// TIA Portal V20 export
// export: Created 2025-12-01T14:56:54.8600917Z, ExportSetting None, DisplayName Totally Integrated Automation Portal, DisplayVersion V20 Update 3, DisplayName TIA Portal Openness, DisplayVersion V20 Update 3, DisplayName TIA Portal Version Control Interface, DisplayVersion V20 Update 3, DisplayName STEP 7 Professional, DisplayVersion V20 Update 3, DisplayName STEP 7 Safety, DisplayVersion V20 Update 2, DisplayName WinCC Basic/Comfort/Advanced, DisplayVersion V20 Update 3, DisplayName WinCC Professional, DisplayVersion V20 Update 3, DisplayName WinCC Unified, DisplayVersion V20 Update 3
FUNCTION_BLOCK "FB343_ApiladorBandejas_RIANTICS"   // FB343, LAD
{ S7_Optimized_Access := 'FALSE' }
// stored: AutoNumber false, SetENOAutomatically false
   VAR_INPUT
      Maquina : UInt;   // Numero de Maquina (Mesa)
      Error_Tx : Bool;   // Error en el Tx
      EnTension : Bool;   // Existe Tension en la Maquina
      MAQx_Desabilitada : Bool;   // Config MAQ. >>> DesHabilitada
      Termico_Elevacion : Bool;   // Termico de la Elevacion
      Pos_DW : Bool;   // Posición Baja del Apilador
      Pos_mid_DW : Bool;
      Pos_mid_UP : Bool;
      Pos_UP : Bool;   // Posición Alta del Apilador
      EnMovimiento_Elevacion : Bool;   // En Movineto la Elevacion
      CargaSuelta : Bool;   // Carga Suelta en el Apilador
      CargaCogida : Bool;   // Carga Cogida en el Apilador
      EnMovimiento_Horquillado : Bool;   // En Movimiento el Hoquillado
      MAQ_DejarBandejas : Bool;   // Interlock >> Dejar Bandejas
      MAQ_CogerBandejas : Bool;   // Interlock >> Coger Bandejas
      MAQ_BuscarCero : Bool;   // Interlock >> Buscar Cero
      CogiendoDerecha : Bool;
      CogiendoIzquierda : Bool;
      DejandoDerecha : Bool;
      DejandoIzquierda : Bool;
      V_TOut_Elevacion : Int := 2000;   // TimeOut del Mov. de Elevacion
      V_TOut_Horquillado : Int := 2000;   // TimeOut del Mov. de Horquillado
   END_VAR
   VAR_OUTPUT
      MAQ_DejadasBandejas : Bool;   // Interlock >> Bandejas Dejadas
      MAQ_CojidasBandejas : Bool;   // Interlock >> Bandejas Cogidas
      MAQ_CeroEncontrado : Bool;   // Interlock >> Bandejas
   END_VAR
   VAR
      AP_ET00 : Bool;
      AP_ET01 : Bool;
      AP_ET100 : Bool;
      AP_ET101 : Bool;
      AP_ET102 : Bool;
      AP_ET103 : Bool;
      AP_ET104 : Bool;
      AP_ET50 : Bool;
      AP_ET51 : Bool;
      AP_ET52 : Bool;
      AP_ET53 : Bool;
      AP_ET54 : Bool;
      AP_ET60 : Bool;
      AP_ET61 : Bool;
      AP_ET62 : Bool;
      AP_ET63 : Bool;
      AP_ET64 : Bool;
      MA_Motor_Elev : Bool;
      MA_Slow_Velocity : Bool;
      MA_CogerCarga : Bool;   // Cerrar Cilindros para coger la pila
      MA_DejarCarga : Bool;   // Abrir Cilindros para dejas la pila
      TMP_ReposoCargaSuelta { S7_SetPoint := 'True'} : TON_TIME;
      TMP_EnTension { S7_SetPoint := 'True'} : "FB910_CNT_UHS";
      TOut_Elevacion { S7_SetPoint := 'True'} : "FB910_CNT_UHS";
      TOut_Horquillado { S7_SetPoint := 'True'} : "FB910_CNT_UHS";
      Manual : "MoviManualMaquina_Apilador_bandejas";
   END_VAR
   VAR_TEMP
      EstadoZona : "EstadoZona";   // Estado de Zona de la Mesa
      EstadoMAQ : "EstadoMaquina_Apilador_bandejas";   // Estado del Vehiculo Inteliguente de la Maquina
      Aux_ET00 : Bool;
   END_VAR
BEGIN

REGION Network 1: INICIALIZAR - Recoger las Variables de Estado de la Maquina
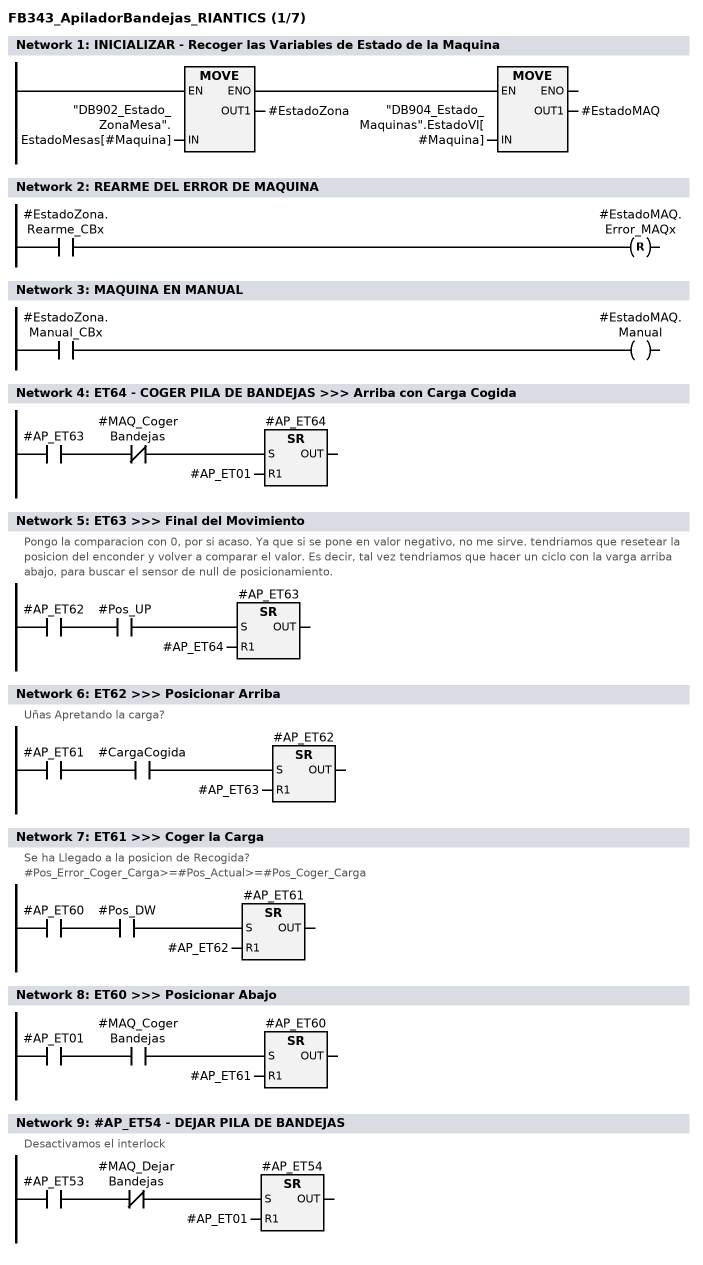
   RUNG wire#powerrail
      Move(in := "DB902_Estado_ZonaMesa".EstadoMesas[#Maquina], out1 => #EstadoZona)
      Move(in := "DB904_Estado_Maquinas".EstadoVI[#Maquina], out1 => #EstadoMAQ)
   END_RUNG
   // the same network as SCL:
   #EstadoZona := "DB902_Estado_ZonaMesa".EstadoMesas[#Maquina];
   #EstadoMAQ := "DB904_Estado_Maquinas".EstadoVI[#Maquina];
END_REGION

REGION Network 2: REARME DEL ERROR DE MAQUINA
   RUNG wire#powerrail
      Contact( #EstadoZona.Rearme_CBx )
      R_Coil( #EstadoMAQ.Error_MAQx )
   END_RUNG
   // the same network as SCL:
   IF #EstadoZona.Rearme_CBx THEN #EstadoMAQ.Error_MAQx := FALSE; END_IF;
END_REGION

REGION Network 3: MAQUINA EN MANUAL
   RUNG wire#powerrail
      Contact( #EstadoZona.Manual_CBx )
      Coil( #EstadoMAQ.Manual )
   END_RUNG
   // the same network as SCL:
   #EstadoMAQ.Manual := #EstadoZona.Manual_CBx;
END_REGION

REGION Network 4: ET64 - COGER PILA DE BANDEJAS >>> Arriba con Carga Cogida
   RUNG wire#powerrail
      Contact( #AP_ET63 )
      I_Contact( #MAQ_CogerBandejas )
      S_SR(operand := #AP_ET64, r1 := #AP_ET01)
   END_RUNG
   // the same network as SCL:
   IF #AP_ET63 AND NOT #MAQ_CogerBandejas THEN
       #AP_ET64 := TRUE;   // SR flip-flop
   END_IF;
   IF #AP_ET01 THEN #AP_ET64 := FALSE; END_IF;
END_REGION

REGION Network 5: ET63 >>> Final del Movimiento
   // Pongo la comparacion con 0, por si acaso. Ya que si se pone en valor negativo, no me sirve. tendriamos que resetear la posicion del enconder y volver a comparar el valor. Es decir, tal vez tendriamos que hacer un ciclo con la varga arriba abajo, para buscar el sensor de null de posicionamiento.
   RUNG wire#powerrail
      Contact( #AP_ET62 )
      Contact( #Pos_UP )
      S_SR(operand := #AP_ET63, r1 := #AP_ET64)
   END_RUNG
   // the same network as SCL:
   IF #AP_ET62 AND #Pos_UP THEN
       #AP_ET63 := TRUE;   // SR flip-flop
   END_IF;
   IF #AP_ET64 THEN #AP_ET63 := FALSE; END_IF;
END_REGION

REGION Network 6: ET62 >>> Posicionar Arriba
   // Uñas Apretando la carga?
   RUNG wire#powerrail
      Contact( #AP_ET61 )
      Contact( #CargaCogida )
      S_SR(operand := #AP_ET62, r1 := #AP_ET63)
   END_RUNG
   // the same network as SCL:
   IF #AP_ET61 AND #CargaCogida THEN
       #AP_ET62 := TRUE;   // SR flip-flop
   END_IF;
   IF #AP_ET63 THEN #AP_ET62 := FALSE; END_IF;
END_REGION

REGION Network 7: ET61 >>> Coger la Carga
   // Se ha Llegado a la posicion de Recogida?
   // #Pos_Error_Coger_Carga>=#Pos_Actual>=#Pos_Coger_Carga
   RUNG wire#powerrail
      Contact( #AP_ET60 )
      Contact( #Pos_DW )
      S_SR(operand := #AP_ET61, r1 := #AP_ET62)
   END_RUNG
   // the same network as SCL:
   IF #AP_ET60 AND #Pos_DW THEN
       #AP_ET61 := TRUE;   // SR flip-flop
   END_IF;
   IF #AP_ET62 THEN #AP_ET61 := FALSE; END_IF;
END_REGION

REGION Network 8: ET60 >>> Posicionar Abajo
   RUNG wire#powerrail
      Contact( #AP_ET01 )
      Contact( #MAQ_CogerBandejas )
      S_SR(operand := #AP_ET60, r1 := #AP_ET61)
   END_RUNG
   // the same network as SCL:
   IF #AP_ET01 AND #MAQ_CogerBandejas THEN
       #AP_ET60 := TRUE;   // SR flip-flop
   END_IF;
   IF #AP_ET61 THEN #AP_ET60 := FALSE; END_IF;
END_REGION

REGION Network 9: #AP_ET54 - DEJAR PILA DE BANDEJAS
   // Desactivamos el interlock
   RUNG wire#powerrail
      Contact( #AP_ET53 )
      I_Contact( #MAQ_DejarBandejas )
      S_SR(operand := #AP_ET54, r1 := #AP_ET01)
   END_RUNG
   // the same network as SCL:
   IF #AP_ET53 AND NOT #MAQ_DejarBandejas THEN
       #AP_ET54 := TRUE;   // SR flip-flop
   END_IF;
   IF #AP_ET01 THEN #AP_ET54 := FALSE; END_IF;
END_REGION

REGION Network 10: ET53 - Bajamos a posicion de espera. para optimizar mov,. apilador esperando>>> abajo con Carga Suelta
   // Coger carga
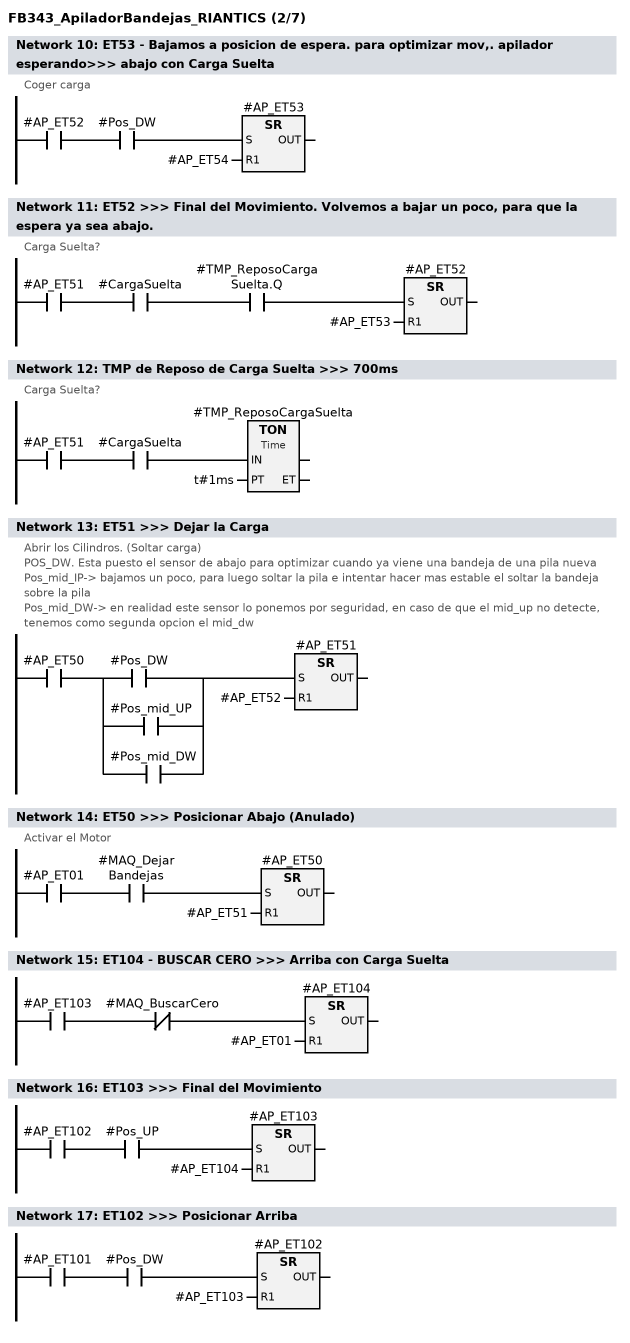
   RUNG wire#powerrail
      Contact( #AP_ET52 )
      Contact( #Pos_DW )
      S_SR(operand := #AP_ET53, r1 := #AP_ET54)
   END_RUNG
   // the same network as SCL:
   IF #AP_ET52 AND #Pos_DW THEN
       #AP_ET53 := TRUE;   // SR flip-flop
   END_IF;
   IF #AP_ET54 THEN #AP_ET53 := FALSE; END_IF;
END_REGION

REGION Network 11: ET52 >>> Final del Movimiento. Volvemos a bajar un poco, para que la espera ya sea abajo.
   // Carga Suelta?
   RUNG wire#powerrail
      Contact( #AP_ET51 )
      Contact( #CargaSuelta )
      Contact( #TMP_ReposoCargaSuelta.Q )
      S_SR(operand := #AP_ET52, r1 := #AP_ET53)
   END_RUNG
   // the same network as SCL:
   IF #AP_ET51 AND #CargaSuelta AND #TMP_ReposoCargaSuelta.Q THEN
       #AP_ET52 := TRUE;   // SR flip-flop
   END_IF;
   IF #AP_ET53 THEN #AP_ET52 := FALSE; END_IF;
END_REGION

REGION Network 12: TMP de Reposo de Carga Suelta >>> 700ms
   // Carga Suelta?
   RUNG wire#powerrail
      Contact( #AP_ET51 )
      Contact( #CargaSuelta )
      { S7_Templates := "time_type := Time" } #TMP_ReposoCargaSuelta.TON(pt := t#1ms, et =>)
   END_RUNG
   // the same network as SCL:
   #TMP_ReposoCargaSuelta(IN := #AP_ET51 AND #CargaSuelta, PT := t#1ms);   // TON
END_REGION

REGION Network 13: ET51 >>> Dejar la Carga
   // Abrir los Cilindros. (Soltar carga)
   // POS_DW. Esta puesto el sensor de abajo para optimizar cuando ya viene una bandeja de una pila nueva
   // Pos_mid_IP-> bajamos un poco, para luego soltar la pila e intentar hacer mas estable el soltar la bandeja sobre la pila
   // Pos_mid_DW-> en realidad este sensor lo ponemos por seguridad, en caso de que el mid_up no detecte, tenemos como segunda opcion el mid_dw
   RUNG wire#powerrail
      Contact( #AP_ET50 )
      wire#w1
      Contact( #Pos_DW )
      wire#w2
      S_SR(operand := #AP_ET51, r1 := #AP_ET52)
   END_RUNG
   RUNG wire#w1
      Contact( #Pos_mid_UP )
   END_RUNG wire#w2
   RUNG wire#w1
      Contact( #Pos_mid_DW )
   END_RUNG wire#w2
   // the same network as SCL:
   IF #AP_ET50 AND (#Pos_DW OR #Pos_mid_UP OR #Pos_mid_DW) THEN
       #AP_ET51 := TRUE;   // SR flip-flop
   END_IF;
   IF #AP_ET52 THEN #AP_ET51 := FALSE; END_IF;
END_REGION

REGION Network 14: ET50 >>> Posicionar Abajo (Anulado)
   // Activar el Motor
   RUNG wire#powerrail
      Contact( #AP_ET01 )
      Contact( #MAQ_DejarBandejas )
      S_SR(operand := #AP_ET50, r1 := #AP_ET51)
   END_RUNG
   // the same network as SCL:
   IF #AP_ET01 AND #MAQ_DejarBandejas THEN
       #AP_ET50 := TRUE;   // SR flip-flop
   END_IF;
   IF #AP_ET51 THEN #AP_ET50 := FALSE; END_IF;
END_REGION

REGION Network 15: ET104 - BUSCAR CERO >>> Arriba con Carga Suelta
   RUNG wire#powerrail
      Contact( #AP_ET103 )
      I_Contact( #MAQ_BuscarCero )
      S_SR(operand := #AP_ET104, r1 := #AP_ET01)
   END_RUNG
   // the same network as SCL:
   IF #AP_ET103 AND NOT #MAQ_BuscarCero THEN
       #AP_ET104 := TRUE;   // SR flip-flop
   END_IF;
   IF #AP_ET01 THEN #AP_ET104 := FALSE; END_IF;
END_REGION

REGION Network 16: ET103 >>> Final del Movimiento
   RUNG wire#powerrail
      Contact( #AP_ET102 )
      Contact( #Pos_UP )
      S_SR(operand := #AP_ET103, r1 := #AP_ET104)
   END_RUNG
   // the same network as SCL:
   IF #AP_ET102 AND #Pos_UP THEN
       #AP_ET103 := TRUE;   // SR flip-flop
   END_IF;
   IF #AP_ET104 THEN #AP_ET103 := FALSE; END_IF;
END_REGION

REGION Network 17: ET102 >>> Posicionar Arriba
   RUNG wire#powerrail
      Contact( #AP_ET101 )
      Contact( #Pos_DW )
      S_SR(operand := #AP_ET102, r1 := #AP_ET103)
   END_RUNG
   // the same network as SCL:
   IF #AP_ET101 AND #Pos_DW THEN
       #AP_ET102 := TRUE;   // SR flip-flop
   END_IF;
   IF #AP_ET103 THEN #AP_ET102 := FALSE; END_IF;
END_REGION

REGION Network 18: ET101 >>> Buscar la Posicion cero (Abajo)
   // Activar el Motor
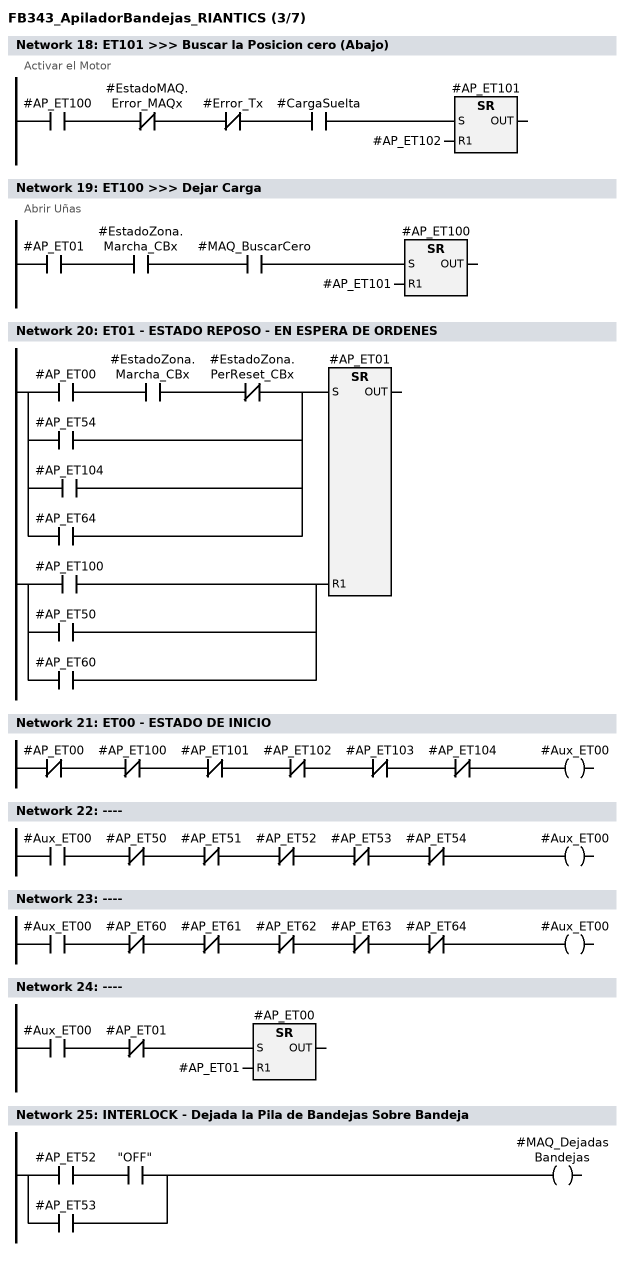
   RUNG wire#powerrail
      Contact( #AP_ET100 )
      I_Contact( #EstadoMAQ.Error_MAQx )
      I_Contact( #Error_Tx )
      Contact( #CargaSuelta )
      S_SR(operand := #AP_ET101, r1 := #AP_ET102)
   END_RUNG
   // the same network as SCL:
   IF #AP_ET100 AND NOT #EstadoMAQ.Error_MAQx AND NOT #Error_Tx AND #CargaSuelta THEN
       #AP_ET101 := TRUE;   // SR flip-flop
   END_IF;
   IF #AP_ET102 THEN #AP_ET101 := FALSE; END_IF;
END_REGION

REGION Network 19: ET100 >>> Dejar Carga
   // Abrir Uñas
   RUNG wire#powerrail
      Contact( #AP_ET01 )
      Contact( #EstadoZona.Marcha_CBx )
      Contact( #MAQ_BuscarCero )
      S_SR(operand := #AP_ET100, r1 := #AP_ET101)
   END_RUNG
   // the same network as SCL:
   IF #AP_ET01 AND #EstadoZona.Marcha_CBx AND #MAQ_BuscarCero THEN
       #AP_ET100 := TRUE;   // SR flip-flop
   END_IF;
   IF #AP_ET101 THEN #AP_ET100 := FALSE; END_IF;
END_REGION

REGION Network 20: ET01 - ESTADO REPOSO - EN ESPERA DE ORDENES
   RUNG wire#powerrail
      Contact( #AP_ET00 )
      Contact( #EstadoZona.Marcha_CBx )
      I_Contact( #EstadoZona.PerReset_CBx )
      wire#w1
      S_SR(operand := #AP_ET01, r1 := wire#w2)
   END_RUNG
   RUNG wire#powerrail
      Contact( #AP_ET54 )
   END_RUNG wire#w1
   RUNG wire#powerrail
      Contact( #AP_ET104 )
   END_RUNG wire#w1
   RUNG wire#powerrail
      Contact( #AP_ET64 )
   END_RUNG wire#w1
   RUNG wire#powerrail
      Contact( #AP_ET100 )
   END_RUNG wire#w2
   RUNG wire#powerrail
      Contact( #AP_ET50 )
   END_RUNG wire#w2
   RUNG wire#powerrail
      Contact( #AP_ET60 )
   END_RUNG wire#w2
   // the same network as SCL:
   IF (#AP_ET00 AND #EstadoZona.Marcha_CBx AND NOT #EstadoZona.PerReset_CBx) OR #AP_ET54 OR #AP_ET104 OR #AP_ET64 THEN
       #AP_ET01 := TRUE;   // SR flip-flop
   END_IF;
   IF #AP_ET100 OR #AP_ET50 OR #AP_ET60 THEN #AP_ET01 := FALSE; END_IF;
END_REGION

REGION Network 21: ET00 - ESTADO DE INICIO
   RUNG wire#powerrail
      I_Contact( #AP_ET00 )
      I_Contact( #AP_ET100 )
      I_Contact( #AP_ET101 )
      I_Contact( #AP_ET102 )
      I_Contact( #AP_ET103 )
      I_Contact( #AP_ET104 )
      Coil( #Aux_ET00 )
   END_RUNG
   // the same network as SCL:
   #Aux_ET00 := NOT #AP_ET00 AND NOT #AP_ET100 AND NOT #AP_ET101 AND NOT #AP_ET102 AND NOT #AP_ET103 AND NOT #AP_ET104;
END_REGION

REGION Network 22: ----
   RUNG wire#powerrail
      Contact( #Aux_ET00 )
      I_Contact( #AP_ET50 )
      I_Contact( #AP_ET51 )
      I_Contact( #AP_ET52 )
      I_Contact( #AP_ET53 )
      I_Contact( #AP_ET54 )
      Coil( #Aux_ET00 )
   END_RUNG
   // the same network as SCL:
   #Aux_ET00 := #Aux_ET00 AND NOT #AP_ET50 AND NOT #AP_ET51 AND NOT #AP_ET52 AND NOT #AP_ET53 AND NOT #AP_ET54;
END_REGION

REGION Network 23: ----
   RUNG wire#powerrail
      Contact( #Aux_ET00 )
      I_Contact( #AP_ET60 )
      I_Contact( #AP_ET61 )
      I_Contact( #AP_ET62 )
      I_Contact( #AP_ET63 )
      I_Contact( #AP_ET64 )
      Coil( #Aux_ET00 )
   END_RUNG
   // the same network as SCL:
   #Aux_ET00 := #Aux_ET00 AND NOT #AP_ET60 AND NOT #AP_ET61 AND NOT #AP_ET62 AND NOT #AP_ET63 AND NOT #AP_ET64;
END_REGION

REGION Network 24: ----
   RUNG wire#powerrail
      Contact( #Aux_ET00 )
      I_Contact( #AP_ET01 )
      S_SR(operand := #AP_ET00, r1 := #AP_ET01)
   END_RUNG
   // the same network as SCL:
   IF #Aux_ET00 AND NOT #AP_ET01 THEN
       #AP_ET00 := TRUE;   // SR flip-flop
   END_IF;
   IF #AP_ET01 THEN #AP_ET00 := FALSE; END_IF;
END_REGION

REGION Network 25: INTERLOCK - Dejada la Pila de Bandejas Sobre Bandeja
   RUNG wire#powerrail
      Contact( #AP_ET52 )
      Contact( "OFF" )
      wire#w1
      Coil( #MAQ_DejadasBandejas )
   END_RUNG
   RUNG wire#powerrail
      Contact( #AP_ET53 )
   END_RUNG wire#w1
   // the same network as SCL:
   #MAQ_DejadasBandejas := (#AP_ET52 AND "OFF") OR #AP_ET53;
END_REGION

REGION Network 26: VARIABLES AUXILIARES - Fin de Reset
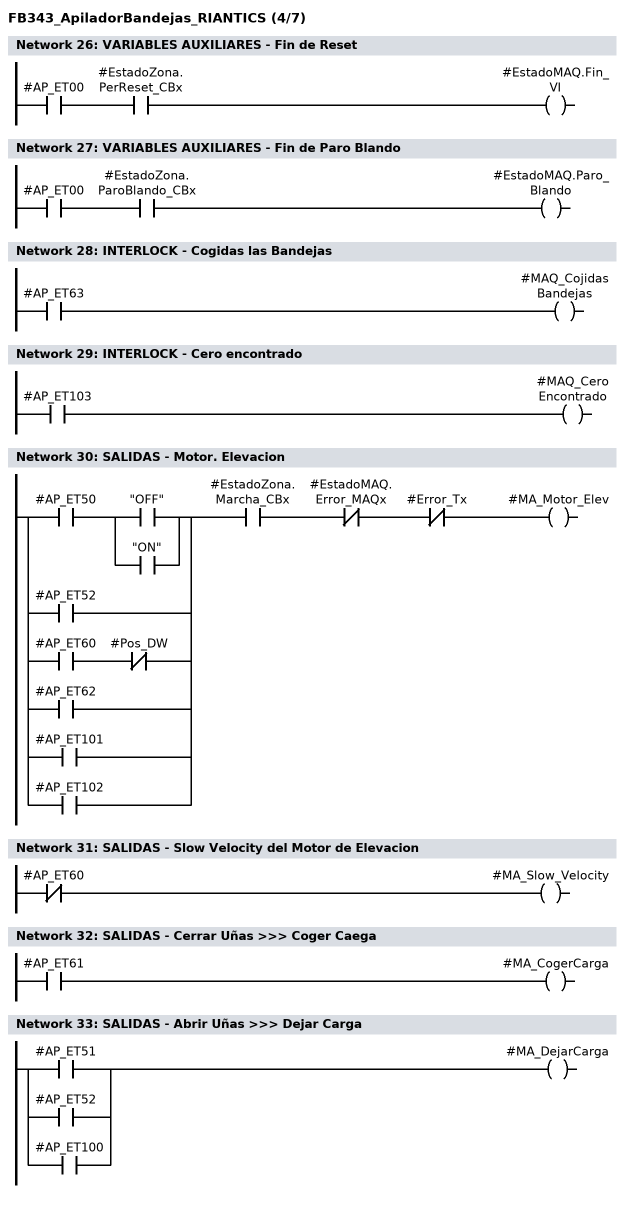
   RUNG wire#powerrail
      Contact( #AP_ET00 )
      Contact( #EstadoZona.PerReset_CBx )
      Coil( #EstadoMAQ.Fin_VI )
   END_RUNG
   // the same network as SCL:
   #EstadoMAQ.Fin_VI := #AP_ET00 AND #EstadoZona.PerReset_CBx;
END_REGION

REGION Network 27: VARIABLES AUXILIARES - Fin de Paro Blando
   RUNG wire#powerrail
      Contact( #AP_ET00 )
      Contact( #EstadoZona.ParoBlando_CBx )
      Coil( #EstadoMAQ.Paro_Blando )
   END_RUNG
   // the same network as SCL:
   #EstadoMAQ.Paro_Blando := #AP_ET00 AND #EstadoZona.ParoBlando_CBx;
END_REGION

REGION Network 28: INTERLOCK - Cogidas las Bandejas
   RUNG wire#powerrail
      Contact( #AP_ET63 )
      Coil( #MAQ_CojidasBandejas )
   END_RUNG
   // the same network as SCL:
   #MAQ_CojidasBandejas := #AP_ET63;
END_REGION

REGION Network 29: INTERLOCK - Cero encontrado
   RUNG wire#powerrail
      Contact( #AP_ET103 )
      Coil( #MAQ_CeroEncontrado )
   END_RUNG
   // the same network as SCL:
   #MAQ_CeroEncontrado := #AP_ET103;
END_REGION

REGION Network 30: SALIDAS - Motor. Elevacion
   RUNG wire#powerrail
      Contact( #AP_ET50 )
      wire#w1
      Contact( "OFF" )
      wire#w2
      Contact( #EstadoZona.Marcha_CBx )
      I_Contact( #EstadoMAQ.Error_MAQx )
      I_Contact( #Error_Tx )
      Coil( #MA_Motor_Elev )
   END_RUNG
   RUNG wire#w1
      Contact( "ON" )
   END_RUNG wire#w2
   RUNG wire#powerrail
      Contact( #AP_ET52 )
   END_RUNG wire#w2
   RUNG wire#powerrail
      Contact( #AP_ET60 )
      I_Contact( #Pos_DW )
   END_RUNG wire#w2
   RUNG wire#powerrail
      Contact( #AP_ET62 )
   END_RUNG wire#w2
   RUNG wire#powerrail
      Contact( #AP_ET101 )
   END_RUNG wire#w2
   RUNG wire#powerrail
      Contact( #AP_ET102 )
   END_RUNG wire#w2
   // the same network as SCL:
   #MA_Motor_Elev := ((#AP_ET50 AND ("OFF" OR "ON")) OR #AP_ET52 OR (#AP_ET60 AND NOT #Pos_DW) OR #AP_ET62 OR #AP_ET101 OR #AP_ET102) AND #EstadoZona.Marcha_CBx AND NOT #EstadoMAQ.Error_MAQx AND NOT #Error_Tx;
END_REGION

REGION Network 31: SALIDAS - Slow Velocity del Motor de Elevacion
   RUNG wire#powerrail
      I_Contact( #AP_ET60 )
      Coil( #MA_Slow_Velocity )
   END_RUNG
   // the same network as SCL:
   #MA_Slow_Velocity := NOT #AP_ET60;
END_REGION

REGION Network 32: SALIDAS - Cerrar Uñas >>> Coger Caega
   RUNG wire#powerrail
      Contact( #AP_ET61 )
      Coil( #MA_CogerCarga )
   END_RUNG
   // the same network as SCL:
   #MA_CogerCarga := #AP_ET61;
END_REGION

REGION Network 33: SALIDAS - Abrir Uñas >>> Dejar Carga
   RUNG wire#powerrail
      Contact( #AP_ET51 )
      wire#w1
      Coil( #MA_DejarCarga )
   END_RUNG
   RUNG wire#powerrail
      Contact( #AP_ET52 )
   END_RUNG wire#w1
   RUNG wire#powerrail
      Contact( #AP_ET100 )
   END_RUNG wire#w1
   // the same network as SCL:
   #MA_DejarCarga := #AP_ET51 OR #AP_ET52 OR #AP_ET100;
END_REGION

REGION Network 34: TMP - Espera En Tension
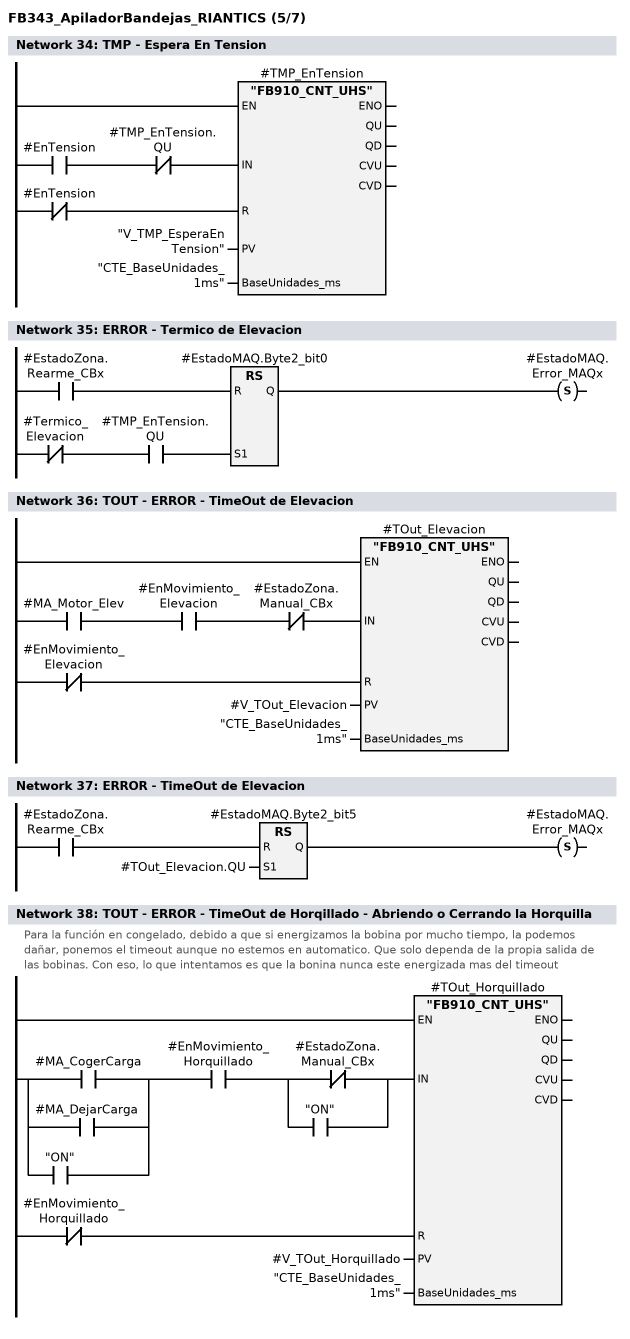
   RUNG wire#powerrail
      #TMP_EnTension(IN := wire#w1, R := wire#w2, PV := "V_TMP_EsperaEnTension", BaseUnidades_ms := "CTE_BaseUnidades_1ms", QU =>, QD =>, CVU =>, CVD =>)
   END_RUNG
   RUNG wire#powerrail
      Contact( #EnTension )
      I_Contact( #TMP_EnTension.QU )
   END_RUNG wire#w1
   RUNG wire#powerrail
      I_Contact( #EnTension )
   END_RUNG wire#w2
   // the same network as SCL:
   #TMP_EnTension(IN := #EnTension AND NOT #TMP_EnTension.QU,   // "FB910_CNT_UHS"
                  R := NOT #EnTension,
                  PV := "V_TMP_EsperaEnTension",
                  BaseUnidades_ms := "CTE_BaseUnidades_1ms");
END_REGION

REGION Network 35: ERROR - Termico de Elevacion
   RUNG wire#powerrail
      Contact( #EstadoZona.Rearme_CBx )
      S_RS(operand := #EstadoMAQ.Byte2_bit0, s1 := wire#w1)
      S_Coil( #EstadoMAQ.Error_MAQx )
   END_RUNG
   RUNG wire#powerrail
      I_Contact( #Termico_Elevacion )
      Contact( #TMP_EnTension.QU )
   END_RUNG wire#w1
   // the same network as SCL:
   IF #EstadoZona.Rearme_CBx THEN
       #EstadoMAQ.Byte2_bit0 := FALSE;   // RS flip-flop
   END_IF;
   IF NOT #Termico_Elevacion AND #TMP_EnTension.QU THEN #EstadoMAQ.Byte2_bit0 := TRUE; END_IF;
   IF #EstadoMAQ.Byte2_bit0 THEN #EstadoMAQ.Error_MAQx := TRUE; END_IF;
END_REGION

REGION Network 36: TOUT - ERROR - TimeOut de Elevacion
   RUNG wire#powerrail
      #TOut_Elevacion(IN := wire#w1, R := wire#w2, PV := #V_TOut_Elevacion, BaseUnidades_ms := "CTE_BaseUnidades_1ms", QU =>, QD =>, CVU =>, CVD =>)
   END_RUNG
   RUNG wire#powerrail
      Contact( #MA_Motor_Elev )
      Contact( #EnMovimiento_Elevacion )
      I_Contact( #EstadoZona.Manual_CBx )
   END_RUNG wire#w1
   RUNG wire#powerrail
      I_Contact( #EnMovimiento_Elevacion )
   END_RUNG wire#w2
   // the same network as SCL:
   #TOut_Elevacion(IN := #MA_Motor_Elev AND #EnMovimiento_Elevacion AND NOT #EstadoZona.Manual_CBx,   // "FB910_CNT_UHS"
                   R := NOT #EnMovimiento_Elevacion,
                   PV := #V_TOut_Elevacion,
                   BaseUnidades_ms := "CTE_BaseUnidades_1ms");
END_REGION

REGION Network 37: ERROR - TimeOut de Elevacion
   RUNG wire#powerrail
      Contact( #EstadoZona.Rearme_CBx )
      S_RS(operand := #EstadoMAQ.Byte2_bit5, s1 := #TOut_Elevacion.QU)
      S_Coil( #EstadoMAQ.Error_MAQx )
   END_RUNG
   // the same network as SCL:
   IF #EstadoZona.Rearme_CBx THEN
       #EstadoMAQ.Byte2_bit5 := FALSE;   // RS flip-flop
   END_IF;
   IF #TOut_Elevacion.QU THEN #EstadoMAQ.Byte2_bit5 := TRUE; END_IF;
   IF #EstadoMAQ.Byte2_bit5 THEN #EstadoMAQ.Error_MAQx := TRUE; END_IF;
END_REGION

REGION Network 38: TOUT - ERROR - TimeOut de Horqillado - Abriendo o Cerrando la Horquilla
   // Para la función en congelado, debido a que si energizamos la bobina por mucho tiempo, la podemos dañar, ponemos el timeout aunque no estemos en automatico. Que solo dependa de la propia salida de las bobinas. Con eso, lo que intentamos es que la bonina nunca este energizada mas del timeout
   RUNG wire#powerrail
      #TOut_Horquillado(IN := wire#w3, R := wire#w4, PV := #V_TOut_Horquillado, BaseUnidades_ms := "CTE_BaseUnidades_1ms", QU =>, QD =>, CVU =>, CVD =>)
   END_RUNG
   RUNG wire#powerrail
      Contact( #MA_CogerCarga )
      wire#w1
      Contact( #EnMovimiento_Horquillado )
      wire#w2
      I_Contact( #EstadoZona.Manual_CBx )
   END_RUNG wire#w3
   RUNG wire#powerrail
      Contact( #MA_DejarCarga )
   END_RUNG wire#w1
   RUNG wire#powerrail
      Contact( "ON" )
   END_RUNG wire#w1
   RUNG wire#w2
      Contact( "ON" )
   END_RUNG wire#w3
   RUNG wire#powerrail
      I_Contact( #EnMovimiento_Horquillado )
   END_RUNG wire#w4
   // the same network as SCL:
   #TOut_Horquillado(IN := (#MA_CogerCarga OR #MA_DejarCarga OR "ON") AND #EnMovimiento_Horquillado AND (NOT #EstadoZona.Manual_CBx OR "ON"),   // "FB910_CNT_UHS"
                     R := NOT #EnMovimiento_Horquillado,
                     PV := #V_TOut_Horquillado,
                     BaseUnidades_ms := "CTE_BaseUnidades_1ms");
END_REGION

REGION Network 39: ERROR - TimeOut de Horqillado - Abriendo la Horquilla
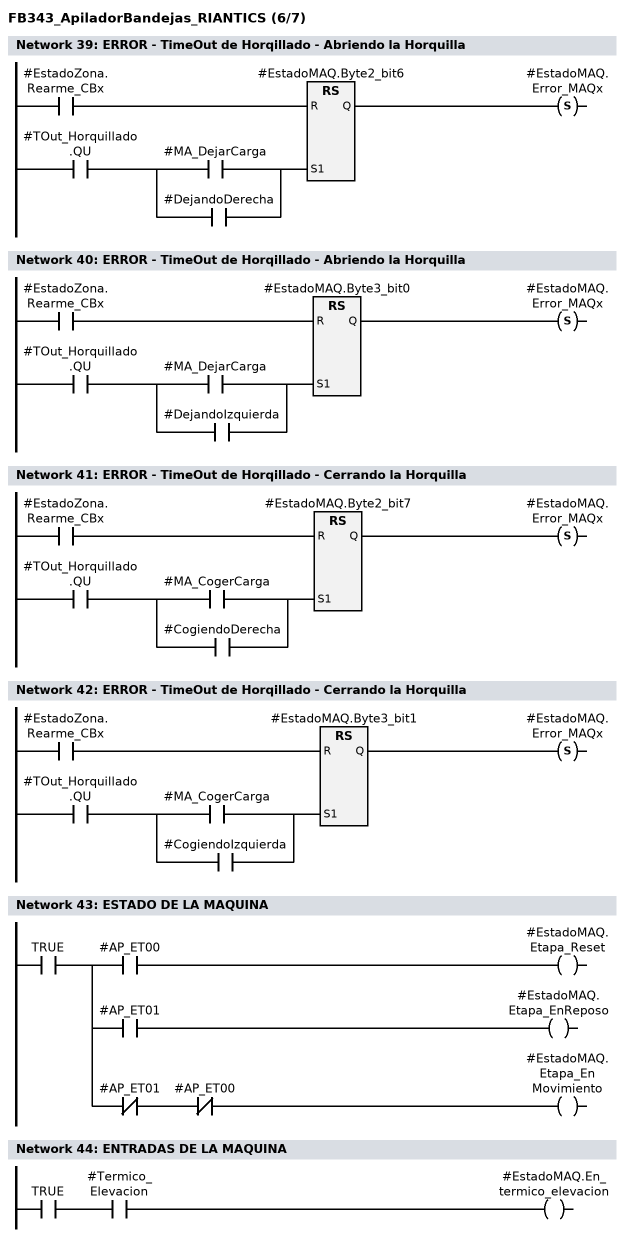
   RUNG wire#powerrail
      Contact( #EstadoZona.Rearme_CBx )
      S_RS(operand := #EstadoMAQ.Byte2_bit6, s1 := wire#w2)
      S_Coil( #EstadoMAQ.Error_MAQx )
   END_RUNG
   RUNG wire#powerrail
      Contact( #TOut_Horquillado.QU )
      wire#w1
      Contact( #MA_DejarCarga )
   END_RUNG wire#w2
   RUNG wire#w1
      Contact( #DejandoDerecha )
   END_RUNG wire#w2
   // the same network as SCL:
   IF #EstadoZona.Rearme_CBx THEN
       #EstadoMAQ.Byte2_bit6 := FALSE;   // RS flip-flop
   END_IF;
   IF #TOut_Horquillado.QU AND (#MA_DejarCarga OR #DejandoDerecha) THEN
       #EstadoMAQ.Byte2_bit6 := TRUE;
   END_IF;
   IF #EstadoMAQ.Byte2_bit6 THEN #EstadoMAQ.Error_MAQx := TRUE; END_IF;
END_REGION

REGION Network 40: ERROR - TimeOut de Horqillado - Abriendo la Horquilla
   RUNG wire#powerrail
      Contact( #EstadoZona.Rearme_CBx )
      S_RS(operand := #EstadoMAQ.Byte3_bit0, s1 := wire#w2)
      S_Coil( #EstadoMAQ.Error_MAQx )
   END_RUNG
   RUNG wire#powerrail
      Contact( #TOut_Horquillado.QU )
      wire#w1
      Contact( #MA_DejarCarga )
   END_RUNG wire#w2
   RUNG wire#w1
      Contact( #DejandoIzquierda )
   END_RUNG wire#w2
   // the same network as SCL:
   IF #EstadoZona.Rearme_CBx THEN
       #EstadoMAQ.Byte3_bit0 := FALSE;   // RS flip-flop
   END_IF;
   IF #TOut_Horquillado.QU AND (#MA_DejarCarga OR #DejandoIzquierda) THEN
       #EstadoMAQ.Byte3_bit0 := TRUE;
   END_IF;
   IF #EstadoMAQ.Byte3_bit0 THEN #EstadoMAQ.Error_MAQx := TRUE; END_IF;
END_REGION

REGION Network 41: ERROR - TimeOut de Horqillado - Cerrando la Horquilla
   RUNG wire#powerrail
      Contact( #EstadoZona.Rearme_CBx )
      S_RS(operand := #EstadoMAQ.Byte2_bit7, s1 := wire#w2)
      S_Coil( #EstadoMAQ.Error_MAQx )
   END_RUNG
   RUNG wire#powerrail
      Contact( #TOut_Horquillado.QU )
      wire#w1
      Contact( #MA_CogerCarga )
   END_RUNG wire#w2
   RUNG wire#w1
      Contact( #CogiendoDerecha )
   END_RUNG wire#w2
   // the same network as SCL:
   IF #EstadoZona.Rearme_CBx THEN
       #EstadoMAQ.Byte2_bit7 := FALSE;   // RS flip-flop
   END_IF;
   IF #TOut_Horquillado.QU AND (#MA_CogerCarga OR #CogiendoDerecha) THEN
       #EstadoMAQ.Byte2_bit7 := TRUE;
   END_IF;
   IF #EstadoMAQ.Byte2_bit7 THEN #EstadoMAQ.Error_MAQx := TRUE; END_IF;
END_REGION

REGION Network 42: ERROR - TimeOut de Horqillado - Cerrando la Horquilla
   RUNG wire#powerrail
      Contact( #EstadoZona.Rearme_CBx )
      S_RS(operand := #EstadoMAQ.Byte3_bit1, s1 := wire#w2)
      S_Coil( #EstadoMAQ.Error_MAQx )
   END_RUNG
   RUNG wire#powerrail
      Contact( #TOut_Horquillado.QU )
      wire#w1
      Contact( #MA_CogerCarga )
   END_RUNG wire#w2
   RUNG wire#w1
      Contact( #CogiendoIzquierda )
   END_RUNG wire#w2
   // the same network as SCL:
   IF #EstadoZona.Rearme_CBx THEN
       #EstadoMAQ.Byte3_bit1 := FALSE;   // RS flip-flop
   END_IF;
   IF #TOut_Horquillado.QU AND (#MA_CogerCarga OR #CogiendoIzquierda) THEN
       #EstadoMAQ.Byte3_bit1 := TRUE;
   END_IF;
   IF #EstadoMAQ.Byte3_bit1 THEN #EstadoMAQ.Error_MAQx := TRUE; END_IF;
END_REGION

REGION Network 43: ESTADO DE LA MAQUINA
   RUNG wire#powerrail
      Contact( TRUE )
      wire#w1
      Contact( #AP_ET00 )
      Coil( #EstadoMAQ.Etapa_Reset )
   END_RUNG
   RUNG wire#w1
      Contact( #AP_ET01 )
      Coil( #EstadoMAQ.Etapa_EnReposo )
   END_RUNG
   RUNG wire#w1
      I_Contact( #AP_ET01 )
      I_Contact( #AP_ET00 )
      Coil( #EstadoMAQ.Etapa_EnMovimiento )
   END_RUNG
   // the same network as SCL:
   #EstadoMAQ.Etapa_Reset := TRUE AND #AP_ET00;
   #EstadoMAQ.Etapa_EnReposo := TRUE AND #AP_ET01;
   #EstadoMAQ.Etapa_EnMovimiento := TRUE AND NOT #AP_ET01 AND NOT #AP_ET00;
END_REGION

REGION Network 44: ENTRADAS DE LA MAQUINA
   RUNG wire#powerrail
      Contact( TRUE )
      Contact( #Termico_Elevacion )
      Coil( #EstadoMAQ.En_termico_elevacion )
   END_RUNG
   // the same network as SCL:
   #EstadoMAQ.En_termico_elevacion := TRUE AND #Termico_Elevacion;
END_REGION

REGION Network 45: ---
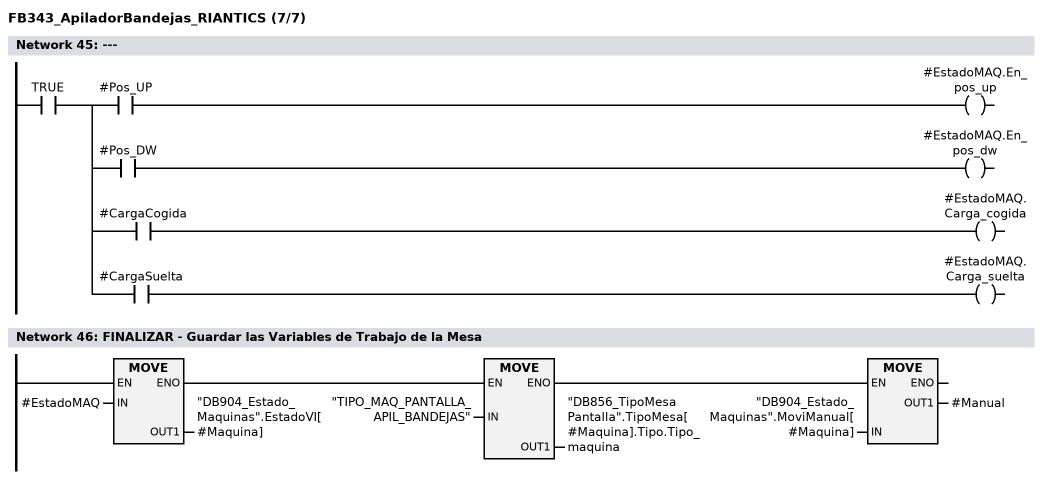
   RUNG wire#powerrail
      Contact( TRUE )
      wire#w1
      Contact( #Pos_UP )
      Coil( #EstadoMAQ.En_pos_up )
   END_RUNG
   RUNG wire#w1
      Contact( #Pos_DW )
      Coil( #EstadoMAQ.En_pos_dw )
   END_RUNG
   RUNG wire#w1
      Contact( #CargaCogida )
      Coil( #EstadoMAQ.Carga_cogida )
   END_RUNG
   RUNG wire#w1
      Contact( #CargaSuelta )
      Coil( #EstadoMAQ.Carga_suelta )
   END_RUNG
   // the same network as SCL:
   #EstadoMAQ.En_pos_up := TRUE AND #Pos_UP;
   #EstadoMAQ.En_pos_dw := TRUE AND #Pos_DW;
   #EstadoMAQ.Carga_cogida := TRUE AND #CargaCogida;
   #EstadoMAQ.Carga_suelta := TRUE AND #CargaSuelta;
END_REGION

REGION Network 46: FINALIZAR - Guardar las Variables de Trabajo de la Mesa
   RUNG wire#powerrail
      Move(in := #EstadoMAQ, out1 => "DB904_Estado_Maquinas".EstadoVI[#Maquina])
      Move(in := "TIPO_MAQ_PANTALLA_APIL_BANDEJAS", out1 => "DB856_TipoMesaPantalla".TipoMesa[#Maquina].Tipo.Tipo_maquina)
      Move(in := "DB904_Estado_Maquinas".MoviManual[#Maquina], out1 => #Manual)
   END_RUNG
   // the same network as SCL:
   "DB904_Estado_Maquinas".EstadoVI[#Maquina] := #EstadoMAQ;
   "DB856_TipoMesaPantalla".TipoMesa[#Maquina].Tipo.Tipo_maquina := "TIPO_MAQ_PANTALLA_APIL_BANDEJAS";
   #Manual := "DB904_Estado_Maquinas".MoviManual[#Maquina];
END_REGION
END_FUNCTION_BLOCK
